FUNCTION_BLOCK TrueUntil (* Generic Actuation / Chain of Actions pattern: move to a position and wait until inPosition becomes true *)
  (* Standard: 61499-2; Description: Copyright (c) 2026 Meisterschulen am Ostbahnhof This program and the accompanying materials are made available under the terms of the Eclipse Public License 2.0 which is available at https://www.eclipse.org/legal/epl-2.0/ SPDX-License-Identifier: EPL-2.0 *)
  (* Version 1.0, 2026-08-31, Franz Höpfinger, Meisterschulen am Ostbahnhof, Generic Actuation / Chain of Actions design pattern (IEC 61499 primer course, Module 6, Valeriy Vyatkin, slides 65-67). REQ treated the same as TRIGGER (re-trigger the move) - the exact intended role of REQ next to TRIGGER on the slide's compact icon is not fully certain, see ChainOfActionsPattern.md *)
  PACKAGE Meins::DesingPatterns::ChainOfActionsPattern;
  (* Documentation:
  Generic, reusable action block for the Generic Actuation / Chain of Actions design patterns (IEC 61499 primer course, Module 6, Valeriy Vyatkin, slides 65-67).
   Same block type for every step of a movement sequence (extend a cylinder, retract a cylinder, slide a workpiece, ...): on TRIGGER (or REQ) it fires TO_POSITION to command the concrete actuator, then waits for inPosition to become TRUE (wired to the actuator's own feedback sensor), then fires STOP and DONE. Chaining several instances via DONE→TRIGGER replaces one large, "spaghetti" ECC covering the whole sequence with a straight-line composition of identical, reusable blocks - see ChainOfActionsPattern.md in this folder for the full write-up, including the demo chain and the open question about the exact role of REQ next to TRIGGER.
  *)
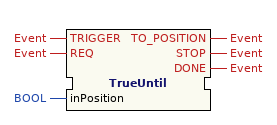
  EVENT_INPUT
    TRIGGER; (* Start moving to the position *)
    REQ; (* Alternate trigger, treated the same as TRIGGER *)
  END_EVENT
  EVENT_OUTPUT
    TO_POSITION; (* Command the actuator to move (wire to the concrete actuator's own move-request event) *)
    STOP; (* Position reached: stop the actuator *)
    DONE; (* Position reached: notify the chain to continue with the next action *)
  END_EVENT
  VAR_INPUT
    inPosition : BOOL; (* TRUE once the actuator has reached the position (wire to the concrete actuator's own feedback sensor) *)
  END_VAR
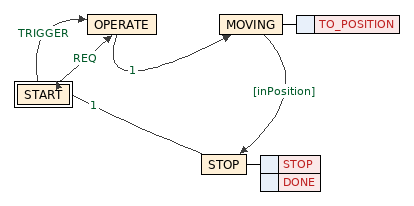
  EC_STATES
    START; (* Idle, waiting for TRIGGER/REQ *)
    OPERATE; (* Triggered, about to move *)
    MOVING : -> TO_POSITION; (* Moving: command the actuator, wait for inPosition *)
    STOP : -> STOP, -> DONE; (* Position reached: stop and report done *)
  END_STATES
  EC_TRANSITIONS
    START TO OPERATE := TRIGGER;
    START TO OPERATE := REQ;
    OPERATE TO MOVING := 1;
    MOVING TO STOP := [inPosition];
    STOP TO START := 1;
  END_TRANSITIONS
END_FUNCTION_BLOCK
